(* Logix 5000 project; controller EuniceF_ICA5 vendor 1 type 14 code 150 rev 37.11; software revision 37.00 *)

TASK MainTask (continuous, watchdog 500 ms) : MainProgram

MODULES
   Local : vendor 1 type 14 code 150 (Compact 0, rev 37.11)
      Discrete_IO : Embedded (Compact 1, rev 3.1, Output RPI 20 ms)
      Analog_IO : Embedded (Compact 2, rev 1.1, Output RPI 80 ms)
      Counters : Embedded (Compact 3, rev 1.1, Output RPI 20 ms)
END_MODULES

VAR_GLOBAL   (* controller tags *)
   COIL1 : ALIAS FOR Local:1:O.Data.2;
   COIL2 : ALIAS FOR Local:1:O.Data.3;
   HIGH : ALIAS FOR Local:1:I.Data.15;
   LOCK : ALIAS FOR Local:1:O.Data.1;
   M1 : ALIAS FOR Local:1:O.Data.0;
   RESET : ALIAS FOR Local:1:I.Data.13;
   START : ALIAS FOR Local:1:I.Data.11;
   STOP : ALIAS FOR Local:1:I.Data.8;
   VIB : ALIAS FOR Local:1:I.Data.14;
END_VAR

PROGRAM MainProgram   (* main routine MainRoutine *)

ROUTINE MainRoutine   (* ladder *)
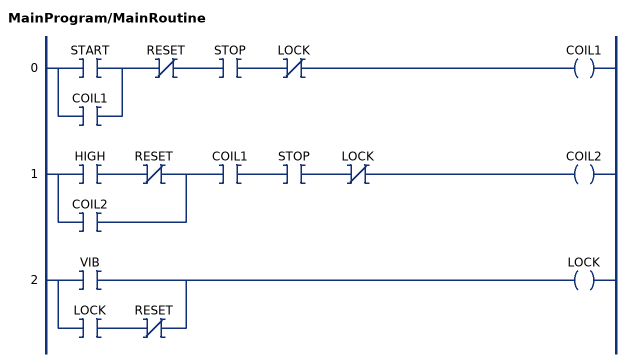
   0: [XIC(START) ,XIC(COIL1) ]XIO(RESET)XIC(STOP)XIO(LOCK)OTE(COIL1);
   1: [XIC(HIGH) XIO(RESET) ,XIC(COIL2) ]XIC(COIL1)XIC(STOP)XIO(LOCK)OTE(COIL2);
   2: [XIC(VIB) ,XIC(LOCK) XIO(RESET) ]OTE(LOCK);
END_ROUTINE
END_PROGRAM
